{attribute 'qualified_only'}
{attribute 'to_string'}
TYPE E_AlarmSeverity :
(
	INFO := 0,
	WARN,
	ERROR
) UINT;
END_TYPE

(* stored: Version 1.1.0.1, ProductVersion 3.1.4026.17
   DUT E_AlarmSeverity: Id {7669db4d-58cd-4116-80e1-3086894cf5fe} *)
